// TIA Portal V17 export
// export: Created 2024-09-02T12:50:26.3604038Z, ExportSetting WithDefaults, DisplayName Totally Integrated Automation Portal, DisplayVersion V17, DisplayName TIA Portal Openness, DisplayVersion V17, DisplayName TIA Portal Version Control Interface, DisplayVersion V17, DisplayName STEP 7 Professional, DisplayVersion V17, DisplayName STEP 7 Safety, DisplayVersion V17, DisplayName WinCC Professional, DisplayVersion V17
TYPE "TypeSeriesError"
// stored: IsFailsafeCompliant false
   STRUCT
      BEA_OK : Bool;
      BEA_NOK : Bool;
      Error_present : Bool;
      HM_Flag : Bool;
      ErrorCounter : Int := 0;
      Para_ErrorNumber : Int := 3;
   END_STRUCT;
END_TYPE
